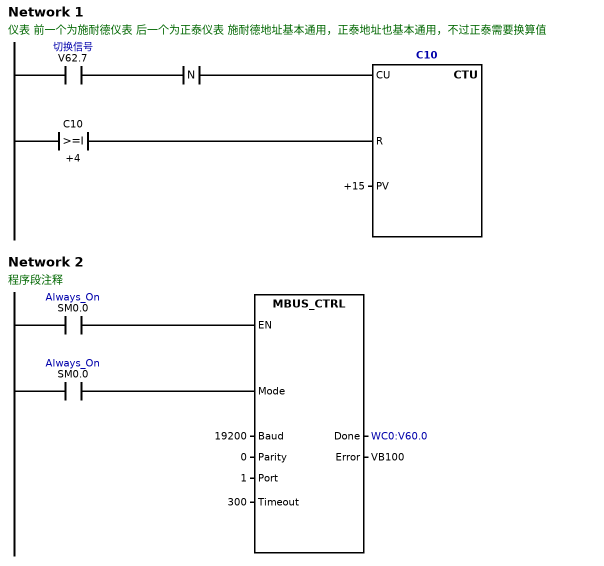
[picture p144: SBR58 networks 1-2]
Network 1
// 仪表 前一个为施耐德仪表 后一个为正泰仪表 施耐德地址基本通用，正泰地址也基本通用，不过正泰需要换算值
LD     切换信号:V62.7
ED
LDW>=  C10, +4
CTU    C10, +15
Network 2
// 程序段注释
LD     Always_On:SM0.0
=      L60.0
LD     Always_On:SM0.0
=      L63.7
LD     L60.0
CALL   MBUS_CTRL:SBR2, L63.7, 19200, 0, 1, 300, WC0:V60.0, VB100
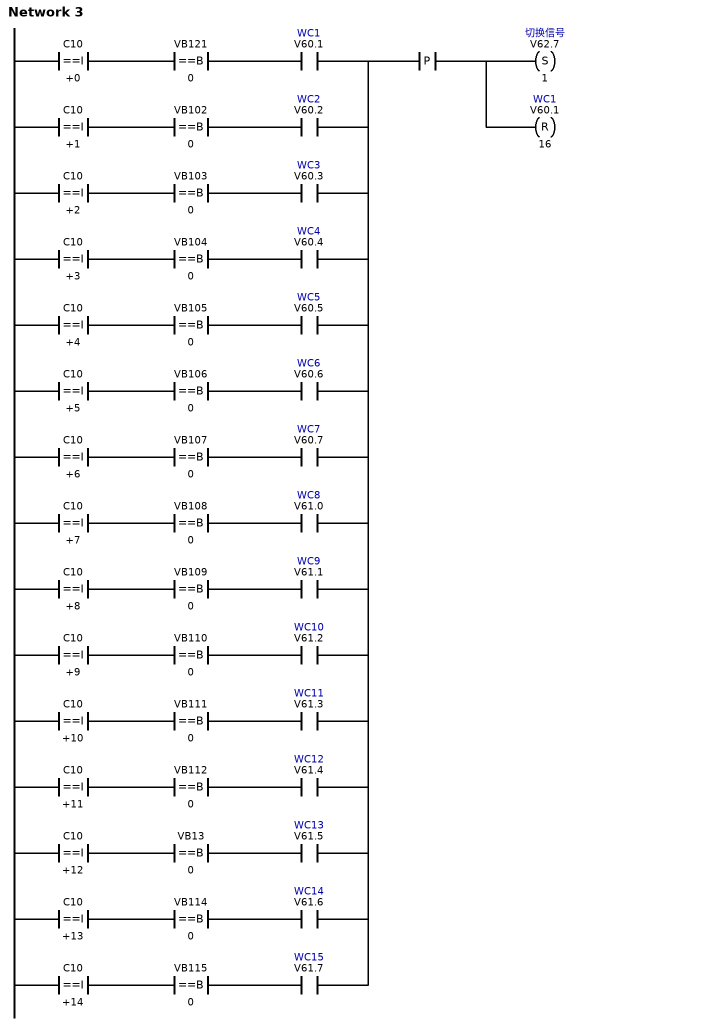
Network 3
LDW=   C10, +0
AB=    VB121, 0
A      WC1:V60.1
LDW=   C10, +1
AB=    VB102, 0
A      WC2:V60.2
OLD
LDW=   C10, +2
AB=    VB103, 0
A      WC3:V60.3
OLD
LDW=   C10, +3
AB=    VB104, 0
A      WC4:V60.4
OLD
LDW=   C10, +4
AB=    VB105, 0
A      WC5:V60.5
OLD
LDW=   C10, +5
AB=    VB106, 0
A      WC6:V60.6
OLD
LDW=   C10, +6
AB=    VB107, 0
A      WC7:V60.7
OLD
LDW=   C10, +7
AB=    VB108, 0
A      WC8:V61.0
OLD
LDW=   C10, +8
AB=    VB109, 0
A      WC9:V61.1
OLD
LDW=   C10, +9
AB=    VB110, 0
A      WC10:V61.2
OLD
LDW=   C10, +10
AB=    VB111, 0
A      WC11:V61.3
OLD
LDW=   C10, +11
AB=    VB112, 0
A      WC12:V61.4
OLD
LDW=   C10, +12
AB=    VB13, 0
A      WC13:V61.5
OLD
LDW=   C10, +13
AB=    VB114, 0
A      WC14:V61.6
OLD
LDW=   C10, +14
AB=    VB115, 0
A      WC15:V61.7
OLD
EU
S      切换信号:V62.7, 1
R      WC1:V60.1, 16
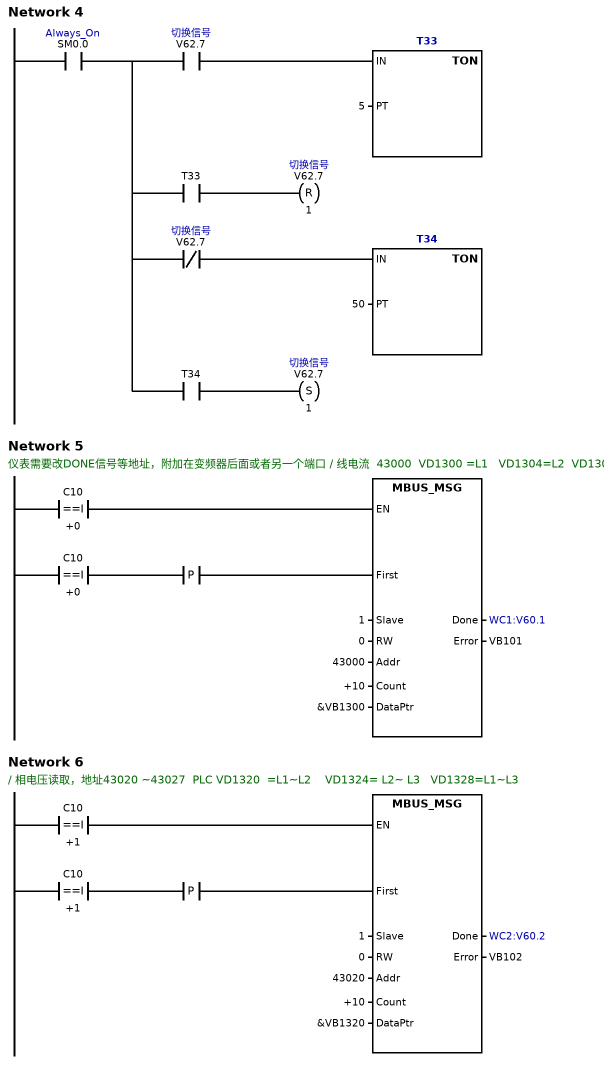
Network 4
LD     Always_On:SM0.0
LPS
A      切换信号:V62.7
TON    T33, 5
LRD
A      T33
R      切换信号:V62.7, 1
LRD
AN     切换信号:V62.7
TON    T34, 50
LPP
A      T34
S      切换信号:V62.7, 1
Network 5
// 仪表需要改DONE信号等地址，附加在变频器后面或者另一个端口
// 线电流  43000  VD1300 =L1   VD1304=L2  VD1308=L3
// 
LDW=   C10, +0
=      L60.0
LDW=   C10, +0
EU
=      L63.7
LD     L60.0
CALL   MBUS_MSG:SBR3, L63.7, 1, 0, 43000, +10, &VB1300, WC1:V60.1, VB101
Network 6
// 
// 相电压读取，地址43020 ~43027  PLC VD1320  =L1~L2    VD1324= L2~ L3   VD1328=L1~L3
LDW=   C10, +1
=      L60.0
LDW=   C10, +1
EU
=      L63.7
LD     L60.0
CALL   MBUS_MSG:SBR3, L63.7, 1, 0, 43020, +10, &VB1320, WC2:V60.2, VB102
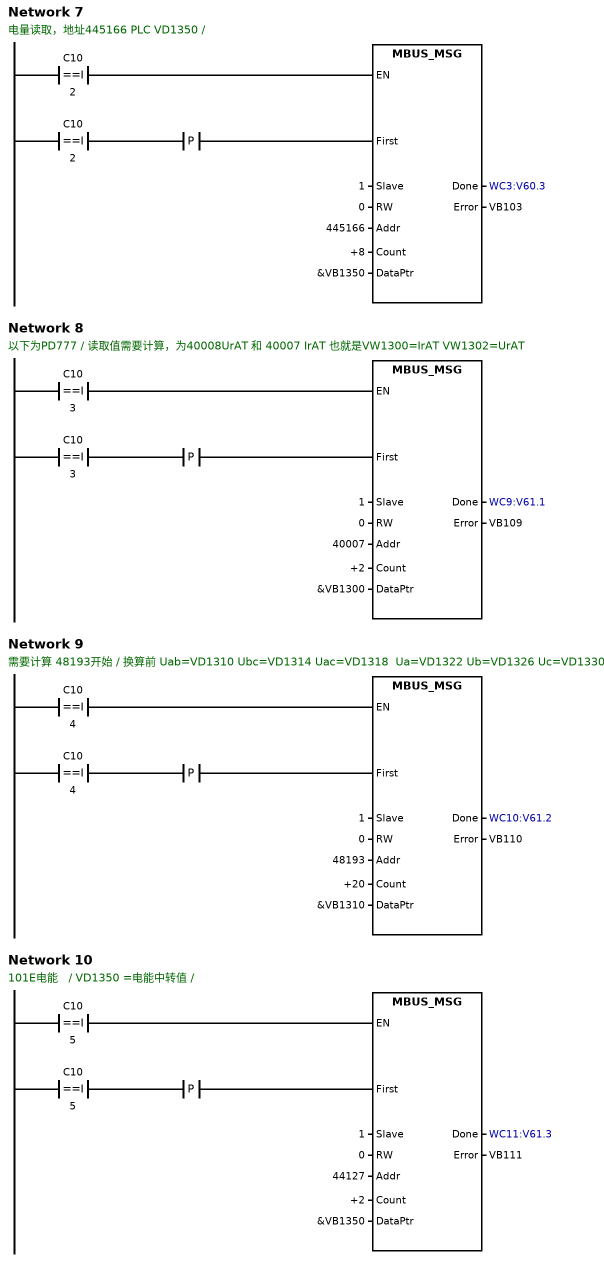
Network 7
// 电量读取，地址445166 PLC VD1350
// 
LDW=   C10, 2
=      L60.0
LDW=   C10, 2
EU
=      L63.7
LD     L60.0
CALL   MBUS_MSG:SBR3, L63.7, 1, 0, 445166, +8, &VB1350, WC3:V60.3, VB103
Network 8
// 以下为PD777
// 读取值需要计算，为40008UrAT 和 40007 IrAT 也就是VW1300=IrAT VW1302=UrAT
LDW=   C10, 3
=      L60.0
LDW=   C10, 3
EU
=      L63.7
LD     L60.0
CALL   MBUS_MSG:SBR3, L63.7, 1, 0, 40007, +2, &VB1300, WC9:V61.1, VB109
Network 9
// 需要计算 48193开始
// 换算前 Uab=VD1310 Ubc=VD1314 Uac=VD1318  Ua=VD1322 Ub=VD1326 Uc=VD1330 
// Ia=VD1334 Ib=VD1338 Ic=VD1342  
// Pt=VD1346 
LDW=   C10, 4
=      L60.0
LDW=   C10, 4
EU
=      L63.7
LD     L60.0
CALL   MBUS_MSG:SBR3, L63.7, 1, 0, 48193, +20, &VB1310, WC10:V61.2, VB110
Network 10
// 101E电能  
// VD1350 =电能中转值
// 
LDW=   C10, 5
=      L60.0
LDW=   C10, 5
EU
=      L63.7
LD     L60.0
CALL   MBUS_MSG:SBR3, L63.7, 1, 0, 44127, +2, &VB1350, WC11:V61.3, VB111
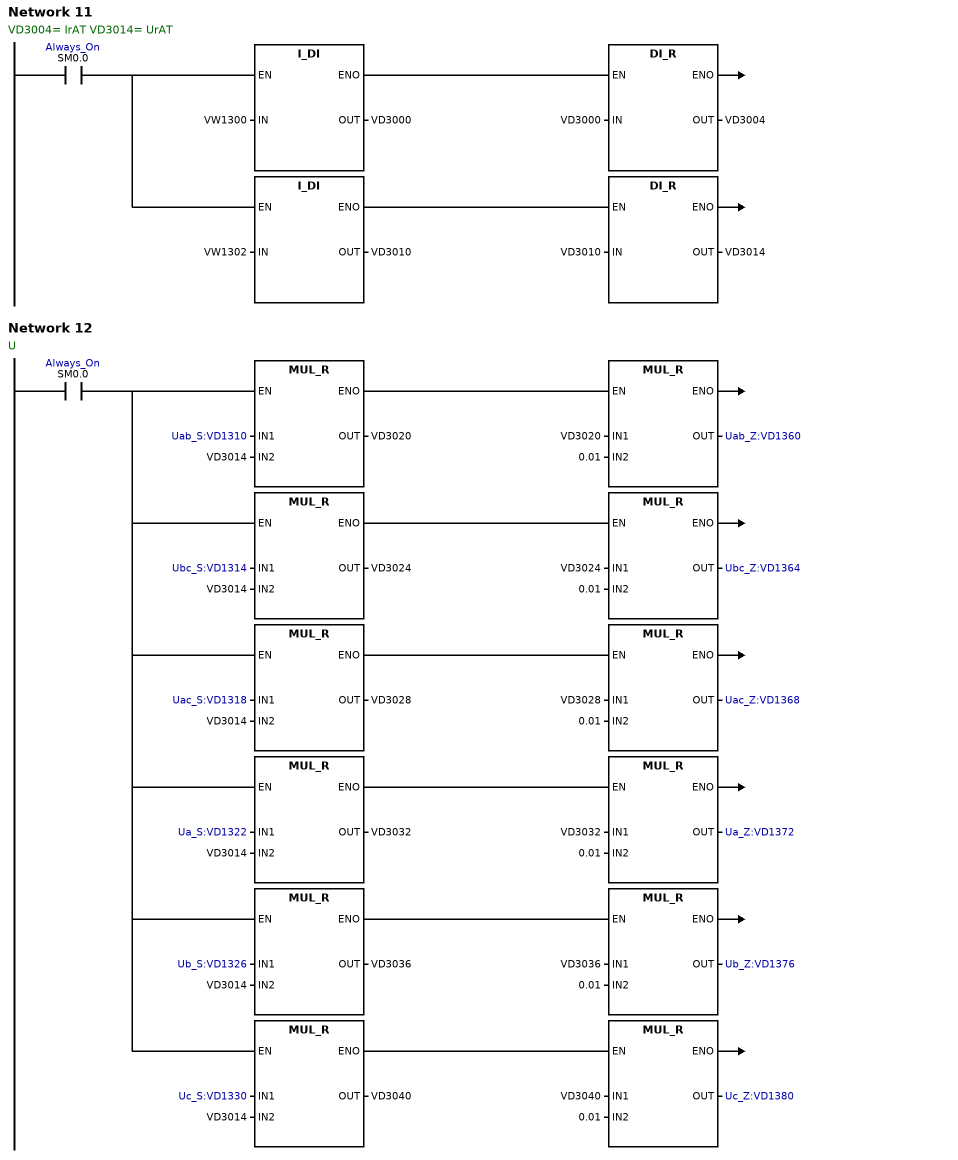
Network 11
// VD3004= IrAT VD3014= UrAT
LD     Always_On:SM0.0
LPS
ITD    VW1300, VD3000
AENO
DTR    VD3000, VD3004
LPP
ITD    VW1302, VD3010
AENO
DTR    VD3010, VD3014
Network 12
// U
LD     Always_On:SM0.0
LPS
MOVR   Uab_S:VD1310, VD3020
AENO
*R     VD3014, VD3020
AENO
MOVR   VD3020, Uab_Z:VD1360
*R     0.01, Uab_Z:VD1360
LRD
MOVR   Ubc_S:VD1314, VD3024
AENO
*R     VD3014, VD3024
AENO
MOVR   VD3024, Ubc_Z:VD1364
*R     0.01, Ubc_Z:VD1364
LRD
MOVR   Uac_S:VD1318, VD3028
AENO
*R     VD3014, VD3028
AENO
MOVR   VD3028, Uac_Z:VD1368
*R     0.01, Uac_Z:VD1368
LRD
MOVR   Ua_S:VD1322, VD3032
AENO
*R     VD3014, VD3032
AENO
MOVR   VD3032, Ua_Z:VD1372
*R     0.01, Ua_Z:VD1372
LRD
MOVR   Ub_S:VD1326, VD3036
AENO
*R     VD3014, VD3036
AENO
MOVR   VD3036, Ub_Z:VD1376
*R     0.01, Ub_Z:VD1376
LPP
MOVR   Uc_S:VD1330, VD3040
AENO
*R     VD3014, VD3040
AENO
MOVR   VD3040, Uc_Z:VD1380
*R     0.01, Uc_Z:VD1380
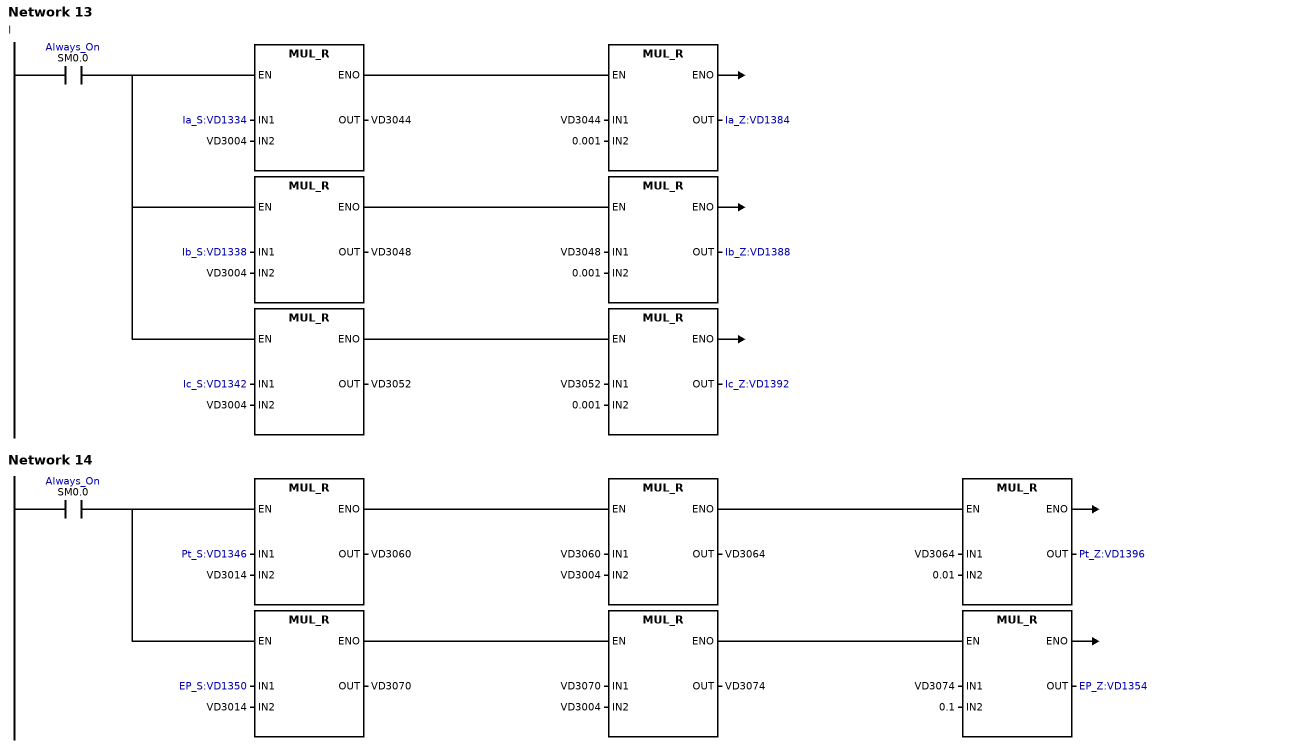
Network 13
// I
LD     Always_On:SM0.0
LPS
MOVR   Ia_S:VD1334, VD3044
AENO
*R     VD3004, VD3044
AENO
MOVR   VD3044, Ia_Z:VD1384
*R     0.001, Ia_Z:VD1384
LRD
MOVR   Ib_S:VD1338, VD3048
AENO
*R     VD3004, VD3048
AENO
MOVR   VD3048, Ib_Z:VD1388
*R     0.001, Ib_Z:VD1388
LPP
MOVR   Ic_S:VD1342, VD3052
AENO
*R     VD3004, VD3052
AENO
MOVR   VD3052, Ic_Z:VD1392
*R     0.001, Ic_Z:VD1392
Network 14
LD     Always_On:SM0.0
LPS
MOVR   Pt_S:VD1346, VD3060
AENO
*R     VD3014, VD3060
AENO
MOVR   VD3060, VD3064
AENO
*R     VD3004, VD3064
AENO
MOVR   VD3064, Pt_Z:VD1396
*R     0.01, Pt_Z:VD1396
LPP
MOVR   EP_S:VD1350, VD3070
AENO
*R     VD3014, VD3070
AENO
MOVR   VD3070, VD3074
AENO
*R     VD3004, VD3074
AENO
MOVR   VD3074, EP_Z:VD1354
*R     0.1, EP_Z:VD1354
END_SUBROUTINE_BLOCK

SUBROUTINE_BLOCK MOD_TCP:SBR60
TITLE=
BEGIN
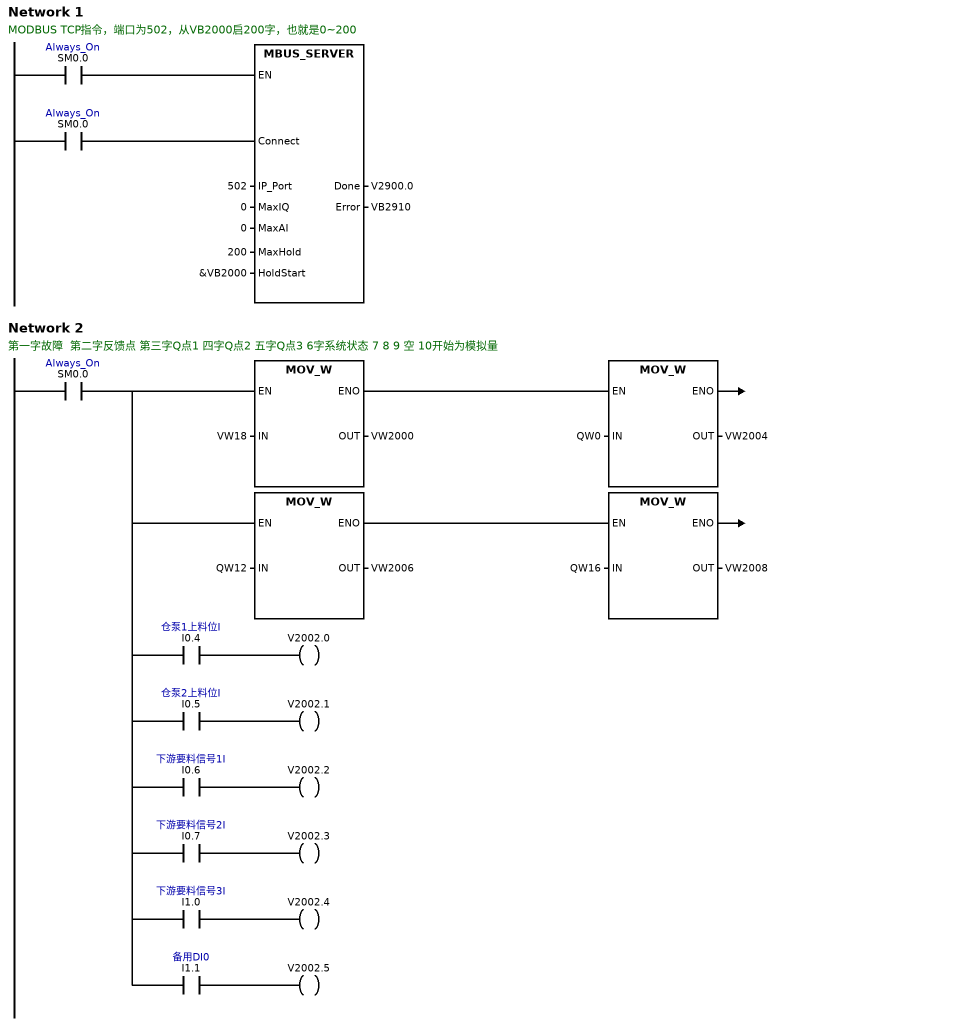
Network 1
// MODBUS TCP指令，端口为502，从VB2000启200字，也就是0~200 
LD     Always_On:SM0.0
=      L60.0
LD     Always_On:SM0.0
=      L63.7
LD     L60.0
CALL   MBUS_SERVER:SBR11, L63.7, 502, 0, 0, 200, &VB2000, V2900.0, VB2910
Network 2
// 第一字故障  第二字反馈点 第三字Q点1 四字Q点2 五字Q点3 6字系统状态 7 8 9 空 10开始为模拟量
LD     Always_On:SM0.0
LPS
MOVW   VW18, VW2000
AENO
MOVW   QW0, VW2004
LRD
MOVW   QW12, VW2006
AENO
MOVW   QW16, VW2008
LRD
A      仓泵1上料位I:I0.4
=      V2002.0
LRD
A      仓泵2上料位I:I0.5
=      V2002.1
LRD
A      下游要料信号1I:I0.6
=      V2002.2
LRD
A      下游要料信号2I:I0.7
=      V2002.3
LRD
A      下游要料信号3I:I1.0
=      V2002.4
LPP
A      备用DI0:I1.1
=      V2002.5
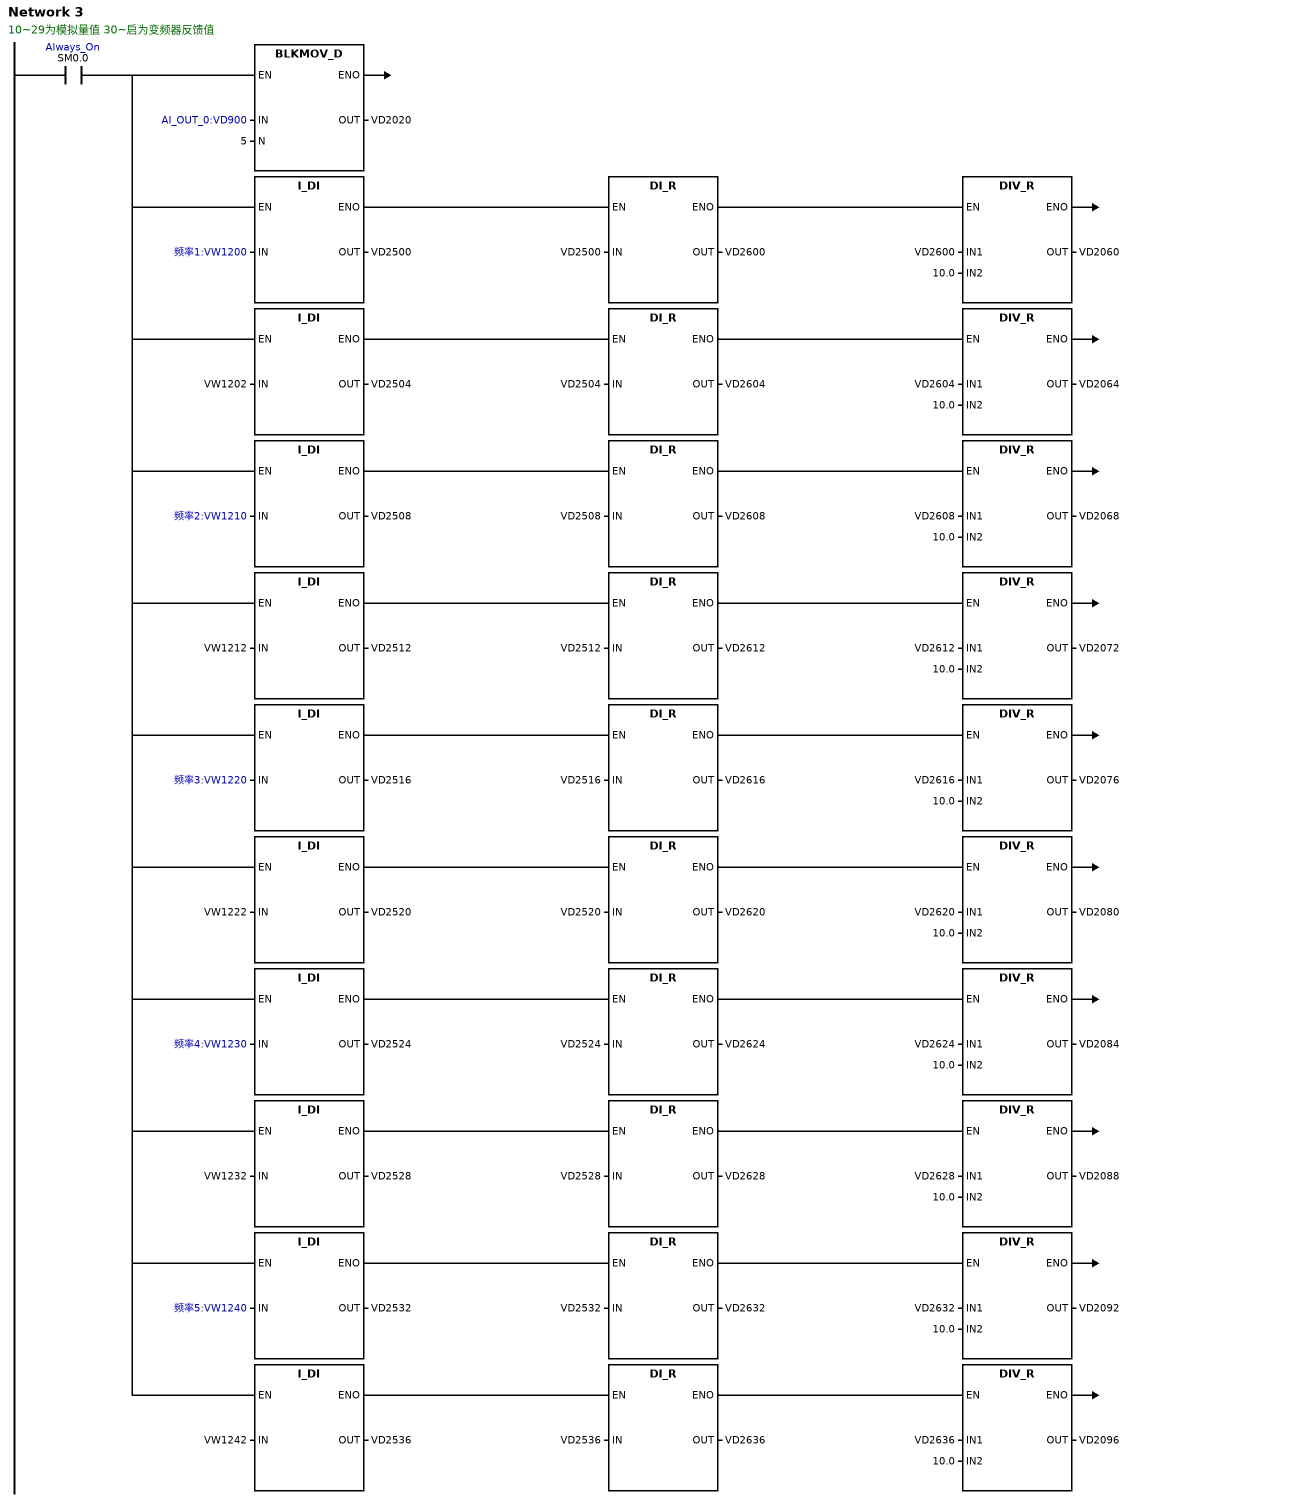
Network 3
// 10~29为模拟量值 30~启为变频器反馈值
LD     Always_On:SM0.0
LPS
BMD    AI_OUT_0:VD900, VD2020, 5
ITD    频率1:VW1200, VD2500
AENO
DTR    VD2500, VD2600
AENO
MOVR   VD2600, VD2060
/R     10.0, VD2060
LRD
ITD    VW1202, VD2504
AENO
DTR    VD2504, VD2604
AENO
MOVR   VD2604, VD2064
/R     10.0, VD2064
LRD
ITD    频率2:VW1210, VD2508
AENO
DTR    VD2508, VD2608
AENO
MOVR   VD2608, VD2068
/R     10.0, VD2068
LRD
ITD    VW1212, VD2512
AENO
DTR    VD2512, VD2612
AENO
MOVR   VD2612, VD2072
/R     10.0, VD2072
LRD
ITD    频率3:VW1220, VD2516
AENO
DTR    VD2516, VD2616
AENO
MOVR   VD2616, VD2076
/R     10.0, VD2076
LRD
ITD    VW1222, VD2520
AENO
DTR    VD2520, VD2620
AENO
MOVR   VD2620, VD2080
/R     10.0, VD2080
LRD
ITD    频率4:VW1230, VD2524
AENO
DTR    VD2524, VD2624
AENO
MOVR   VD2624, VD2084
/R     10.0, VD2084
LRD
ITD    VW1232, VD2528
AENO
DTR    VD2528, VD2628
AENO
MOVR   VD2628, VD2088
/R     10.0, VD2088
LRD
ITD    频率5:VW1240, VD2532
AENO
DTR    VD2532, VD2632
AENO
MOVR   VD2632, VD2092
/R     10.0, VD2092
LPP
ITD    VW1242, VD2536
AENO
DTR    VD2536, VD2636
AENO
MOVR   VD2636, VD2096
/R     10.0, VD2096
END_SUBROUTINE_BLOCK

SUBROUTINE_BLOCK MOD_RTU:SBR61
TITLE=
BEGIN
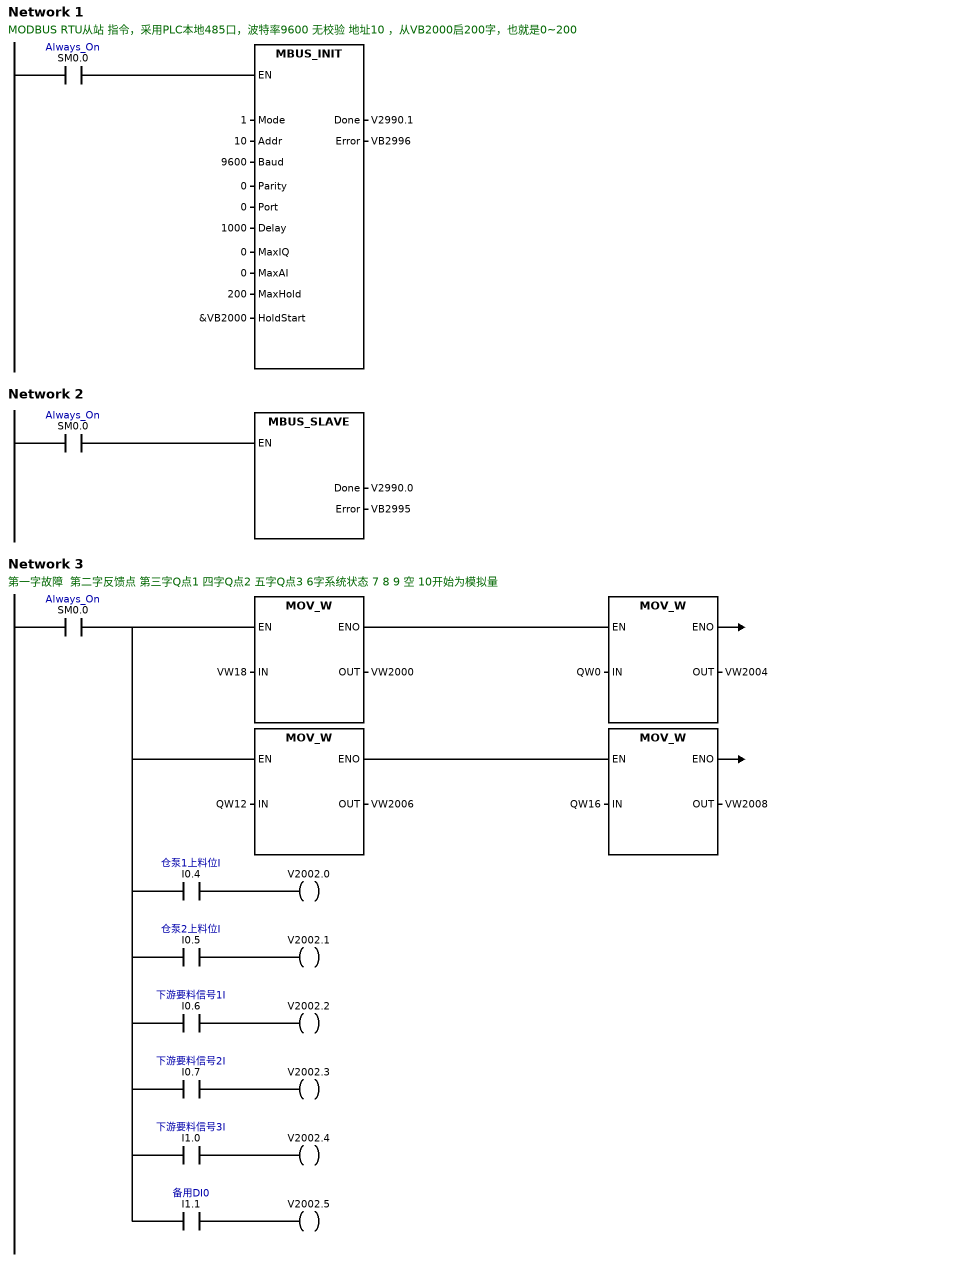
Network 1
// MODBUS RTU从站 指令，采用PLC本地485口，波特率9600 无校验 地址10 ，从VB2000启200字，也就是0~200 
LD     Always_On:SM0.0
CALL   MBUS_INIT:SBR0, 1, 10, 9600, 0, 0, 1000, 0, 0, 200, &VB2000, V2990.1, VB2996
Network 2
LD     Always_On:SM0.0
CALL   MBUS_SLAVE:SBR1, V2990.0, VB2995
Network 3
// 第一字故障  第二字反馈点 第三字Q点1 四字Q点2 五字Q点3 6字系统状态 7 8 9 空 10开始为模拟量
LD     Always_On:SM0.0
LPS
MOVW   VW18, VW2000
AENO
MOVW   QW0, VW2004
LRD
MOVW   QW12, VW2006
AENO
MOVW   QW16, VW2008
LRD
A      仓泵1上料位I:I0.4
=      V2002.0
LRD
A      仓泵2上料位I:I0.5
=      V2002.1
LRD
A      下游要料信号1I:I0.6
=      V2002.2
LRD
A      下游要料信号2I:I0.7
=      V2002.3
LRD
A      下游要料信号3I:I1.0
=      V2002.4
LPP
A      备用DI0:I1.1
=      V2002.5
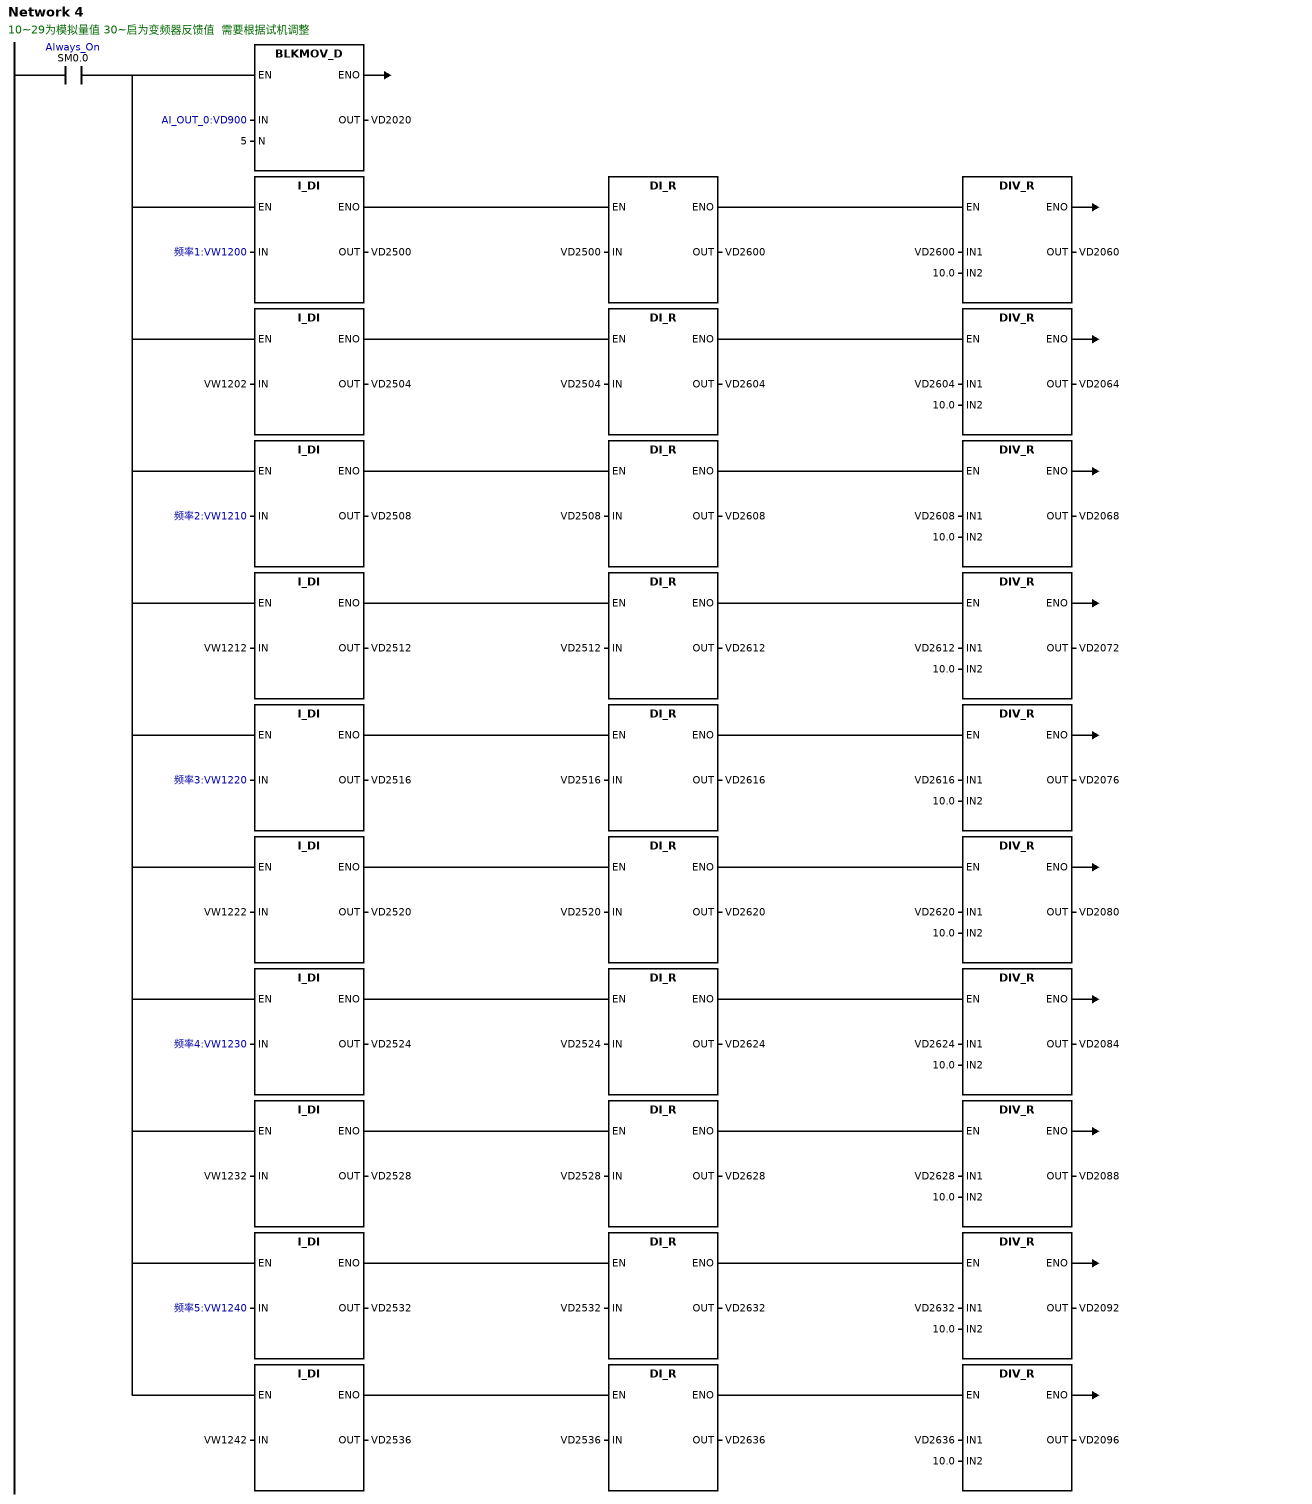
Network 4
// 10~29为模拟量值 30~启为变频器反馈值  需要根据试机调整
LD     Always_On:SM0.0
LPS
BMD    AI_OUT_0:VD900, VD2020, 5
ITD    频率1:VW1200, VD2500
AENO
DTR    VD2500, VD2600
AENO
MOVR   VD2600, VD2060
/R     10.0, VD2060
LRD
ITD    VW1202, VD2504
AENO
DTR    VD2504, VD2604
AENO
MOVR   VD2604, VD2064
/R     10.0, VD2064
LRD
ITD    频率2:VW1210, VD2508
AENO
DTR    VD2508, VD2608
AENO
MOVR   VD2608, VD2068
/R     10.0, VD2068
LRD
ITD    VW1212, VD2512
AENO
DTR    VD2512, VD2612
AENO
MOVR   VD2612, VD2072
/R     10.0, VD2072
LRD
ITD    频率3:VW1220, VD2516
AENO
DTR    VD2516, VD2616
AENO
MOVR   VD2616, VD2076
/R     10.0, VD2076
LRD
ITD    VW1222, VD2520
AENO
DTR    VD2520, VD2620
AENO
MOVR   VD2620, VD2080
/R     10.0, VD2080
LRD
ITD    频率4:VW1230, VD2524
AENO
DTR    VD2524, VD2624
AENO
MOVR   VD2624, VD2084
/R     10.0, VD2084
LRD
ITD    VW1232, VD2528
AENO
DTR    VD2528, VD2628
AENO
MOVR   VD2628, VD2088
/R     10.0, VD2088
LRD
ITD    频率5:VW1240, VD2532
AENO
DTR    VD2532, VD2632
AENO
MOVR   VD2632, VD2092
/R     10.0, VD2092
LPP
ITD    VW1242, VD2536
AENO
DTR    VD2536, VD2636
AENO
MOVR   VD2636, VD2096
/R     10.0, VD2096
END_SUBROUTINE_BLOCK

SUBROUTINE_BLOCK 引风机1:SBR70
TITLE=
VAR_INPUT
IN_SD:BOOL;	// L0.0 
IN_ZD:BOOL;	// L0.1 
IN_Error:BOOL;	// L0.2 
IN_Run_Time:INT;	// LW1 
END_VAR
VAR_OUTPUT
OUT_主:BOOL;	// L3.0  先主
OUT_角:BOOL;	// L3.1 后角
OUT_星:BOOL;	// L3.2 先星
END_VAR
VAR
TP1:BOOL;	// L3.3 
TP2:BOOL;	// L3.4 
END_VAR
BEGIN
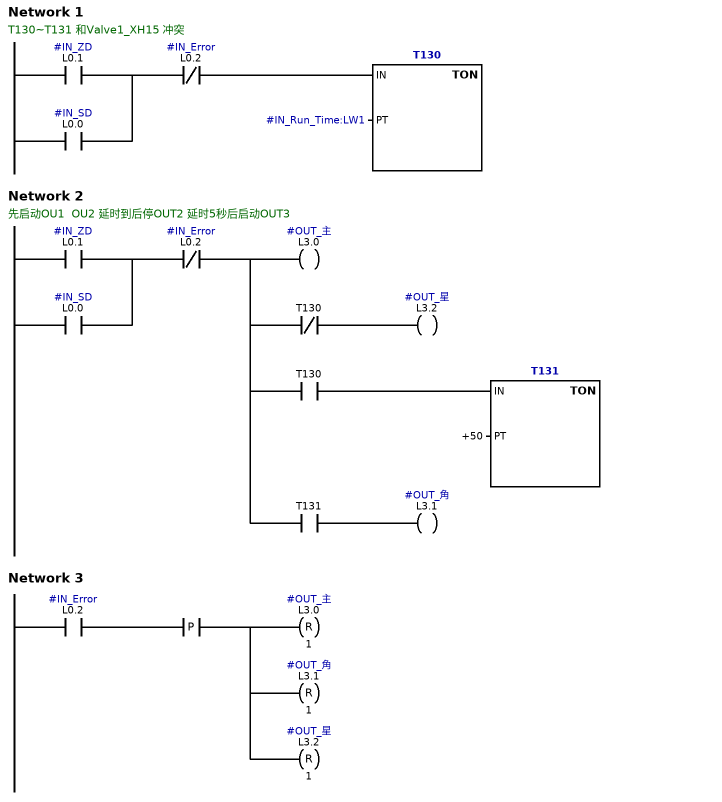
Network 1
// T130~T131 和Valve1_XH15 冲突
LD     #IN_ZD:L0.1
O      #IN_SD:L0.0
AN     #IN_Error:L0.2
TON    T130, #IN_Run_Time:LW1
Network 2
// 先启动OU1  OU2 延时到后停OUT2 延时5秒后启动OUT3
LD     #IN_ZD:L0.1
O      #IN_SD:L0.0
AN     #IN_Error:L0.2
LPS
=      #OUT_主:L3.0
AN     T130
=      #OUT_星:L3.2
LRD
A      T130
TON    T131, +50
LPP
A      T131
=      #OUT_角:L3.1
Network 3
LD     #IN_Error:L0.2
EU
R      #OUT_主:L3.0, 1
R      #OUT_角:L3.1, 1
R      #OUT_星:L3.2, 1
END_SUBROUTINE_BLOCK

SUBROUTINE_BLOCK 引风机2:SBR71
TITLE=
VAR_INPUT
IN_SD:BOOL;	// L0.0 
IN_ZD:BOOL;	// L0.1 
IN_Error:BOOL;	// L0.2 
IN_Run_Time:INT;	// LW1 
END_VAR
VAR_OUTPUT
OUT_ONE1:BOOL;	// L3.0 
OUT_ONE2:BOOL;	// L3.1 
OUT_ONE3:BOOL;	// L3.2 
END_VAR
VAR
TP1:BOOL;	// L3.3 
TP2:BOOL;	// L3.4 
END_VAR
BEGIN
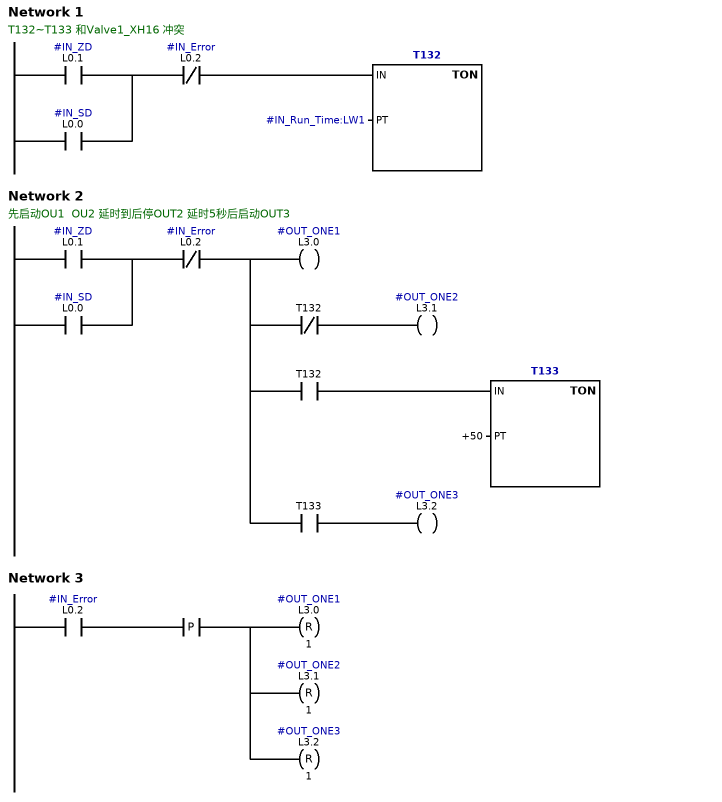
Network 1
// T132~T133 和Valve1_XH16 冲突
LD     #IN_ZD:L0.1
O      #IN_SD:L0.0
AN     #IN_Error:L0.2
TON    T132, #IN_Run_Time:LW1
Network 2
// 先启动OU1  OU2 延时到后停OUT2 延时5秒后启动OUT3
LD     #IN_ZD:L0.1
O      #IN_SD:L0.0
AN     #IN_Error:L0.2
LPS
=      #OUT_ONE1:L3.0
AN     T132
=      #OUT_ONE2:L3.1
LRD
A      T132
TON    T133, +50
LPP
A      T133
=      #OUT_ONE3:L3.2
Network 3
LD     #IN_Error:L0.2
EU
R      #OUT_ONE1:L3.0, 1
R      #OUT_ONE2:L3.1, 1
R      #OUT_ONE3:L3.2, 1
END_SUBROUTINE_BLOCK

SUBROUTINE_BLOCK 引风机3:SBR72
TITLE=
VAR_INPUT
IN_SD:BOOL;	// L0.0 
IN_ZD:BOOL;	// L0.1 
IN_Error:BOOL;	// L0.2 
IN_Run_Time:INT;	// LW1 
END_VAR
VAR_OUTPUT
OUT_ONE1:BOOL;	// L3.0 
OUT_ONE2:BOOL;	// L3.1 
OUT_ONE3:BOOL;	// L3.2 
END_VAR
VAR
TP1:BOOL;	// L3.3 
TP2:BOOL;	// L3.4 
END_VAR
BEGIN
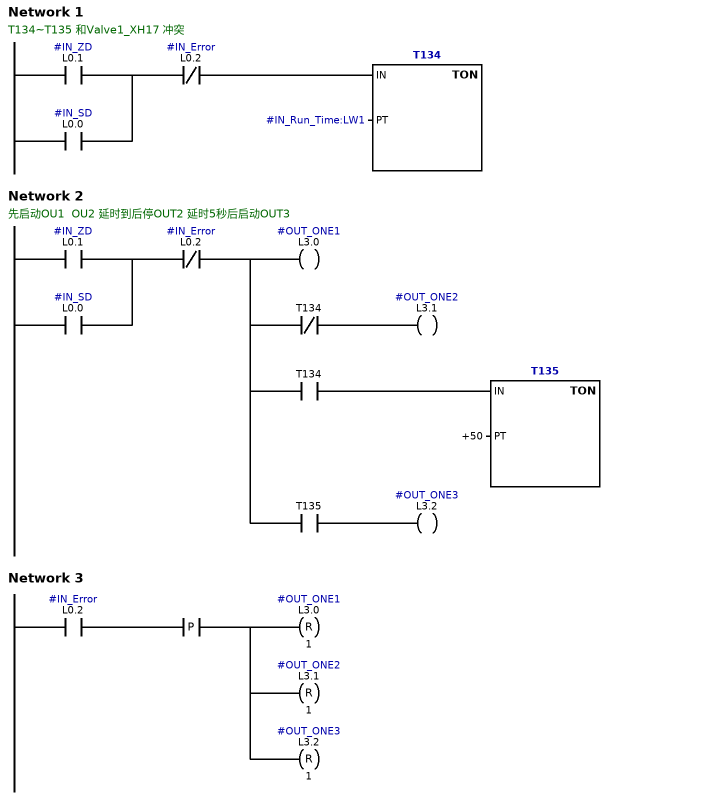
Network 1
// T134~T135 和Valve1_XH17 冲突
LD     #IN_ZD:L0.1
O      #IN_SD:L0.0
AN     #IN_Error:L0.2
TON    T134, #IN_Run_Time:LW1
Network 2
// 先启动OU1  OU2 延时到后停OUT2 延时5秒后启动OUT3
LD     #IN_ZD:L0.1
O      #IN_SD:L0.0
AN     #IN_Error:L0.2
LPS
=      #OUT_ONE1:L3.0
AN     T134
=      #OUT_ONE2:L3.1
LRD
A      T134
TON    T135, +50
LPP
A      T135
=      #OUT_ONE3:L3.2
Network 3
LD     #IN_Error:L0.2
EU
R      #OUT_ONE1:L3.0, 1
R      #OUT_ONE2:L3.1, 1
R      #OUT_ONE3:L3.2, 1
END_SUBROUTINE_BLOCK

SUBROUTINE_BLOCK 引风机4:SBR73
TITLE=
VAR_INPUT
IN_SD:BOOL;	// L0.0 
IN_ZD:BOOL;	// L0.1 
IN_Error:BOOL;	// L0.2 
IN_Run_Time:INT;	// LW1 
END_VAR
VAR_OUTPUT
OUT_ONE1:BOOL;	// L3.0 
OUT_ONE2:BOOL;	// L3.1 
OUT_ONE3:BOOL;	// L3.2 
END_VAR
VAR
TP1:BOOL;	// L3.3 
TP2:BOOL;	// L3.4 
END_VAR
BEGIN
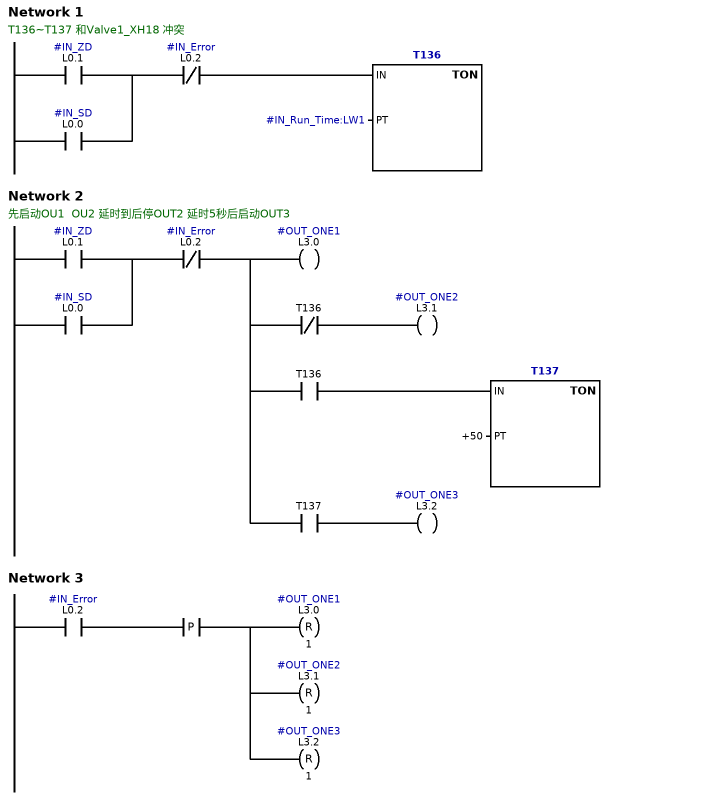
Network 1
// T136~T137 和Valve1_XH18 冲突
LD     #IN_ZD:L0.1
O      #IN_SD:L0.0
AN     #IN_Error:L0.2
TON    T136, #IN_Run_Time:LW1
Network 2
// 先启动OU1  OU2 延时到后停OUT2 延时5秒后启动OUT3
LD     #IN_ZD:L0.1
O      #IN_SD:L0.0
AN     #IN_Error:L0.2
LPS
=      #OUT_ONE1:L3.0
AN     T136
=      #OUT_ONE2:L3.1
LRD
A      T136
TON    T137, +50
LPP
A      T137
=      #OUT_ONE3:L3.2
Network 3
LD     #IN_Error:L0.2
EU
R      #OUT_ONE1:L3.0, 1
R      #OUT_ONE2:L3.1, 1
R      #OUT_ONE3:L3.2, 1
END_SUBROUTINE_BLOCK

SUBROUTINE_BLOCK 引风机5:SBR74
TITLE=
VAR_INPUT
IN_SD:BOOL;	// L0.0 
IN_ZD:BOOL;	// L0.1 
IN_Error:BOOL;	// L0.2 
IN_Run_Time:INT;	// LW1 
END_VAR
VAR_OUTPUT
OUT_ONE1:BOOL;	// L3.0 
OUT_ONE2:BOOL;	// L3.1 
OUT_ONE3:BOOL;	// L3.2 
END_VAR
VAR
TP1:BOOL;	// L3.3 
TP2:BOOL;	// L3.4 
END_VAR
BEGIN
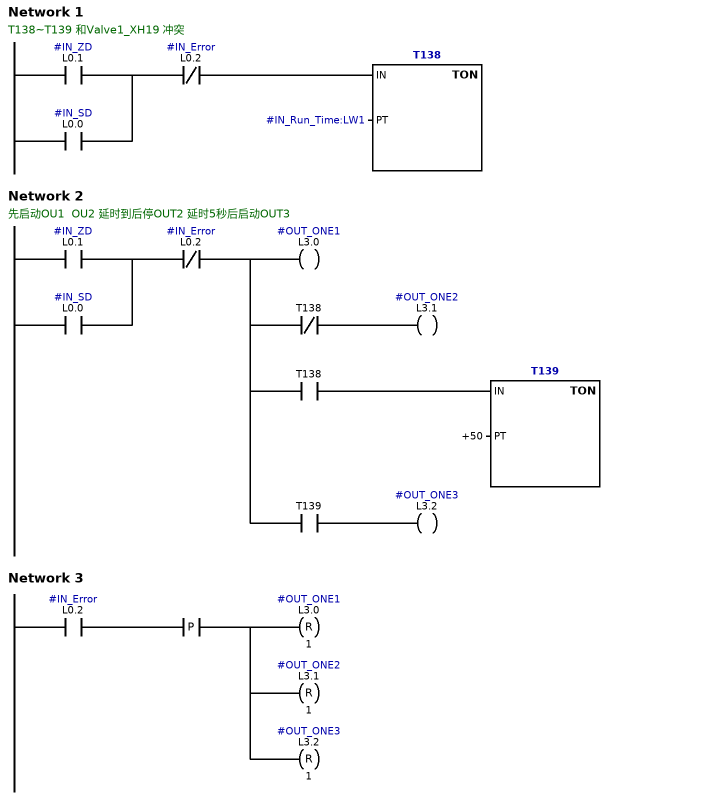
Network 1
// T138~T139 和Valve1_XH19 冲突
LD     #IN_ZD:L0.1
O      #IN_SD:L0.0
AN     #IN_Error:L0.2
TON    T138, #IN_Run_Time:LW1
Network 2
// 先启动OU1  OU2 延时到后停OUT2 延时5秒后启动OUT3
LD     #IN_ZD:L0.1
O      #IN_SD:L0.0
AN     #IN_Error:L0.2
LPS
=      #OUT_ONE1:L3.0
AN     T138
=      #OUT_ONE2:L3.1
LRD
A      T138
TON    T139, +50
LPP
A      T139
=      #OUT_ONE3:L3.2
Network 3
LD     #IN_Error:L0.2
EU
R      #OUT_ONE1:L3.0, 1
R      #OUT_ONE2:L3.1, 1
R      #OUT_ONE3:L3.2, 1
END_SUBROUTINE_BLOCK

SUBROUTINE_BLOCK 除铁器6组4:SBR76
TITLE=
VAR_INPUT
IN_SD:BOOL;	// L0.0 
IN_ZD:BOOL;	// L0.1 
IN_Error:BOOL;	// L0.2 
IN_Run_Time:INT;	// LW1 
IN_Stop_Time:INT;	// LW3 
IN_JG:INT;	// LW5 除铁到排渣间隔
IN_PZ_RT:INT;	// LW7 排渣运行
IN_PZ_ST:INT;	// LW9 排渣间隔
Z_Time:DINT;	// LD11 
END_VAR
VAR_OUTPUT
OUT_1:BOOL;	// L15.0 
OUT_2:BOOL;	// L15.1 
OUT_3:BOOL;	// L15.2 
OUT_4:BOOL;	// L15.3 
OUT_5:BOOL;	// L15.4 
OUT_6:BOOL;	// L15.5 
ZTXH:BOOL;	// L15.6 暂停信号
END_VAR
BEGIN
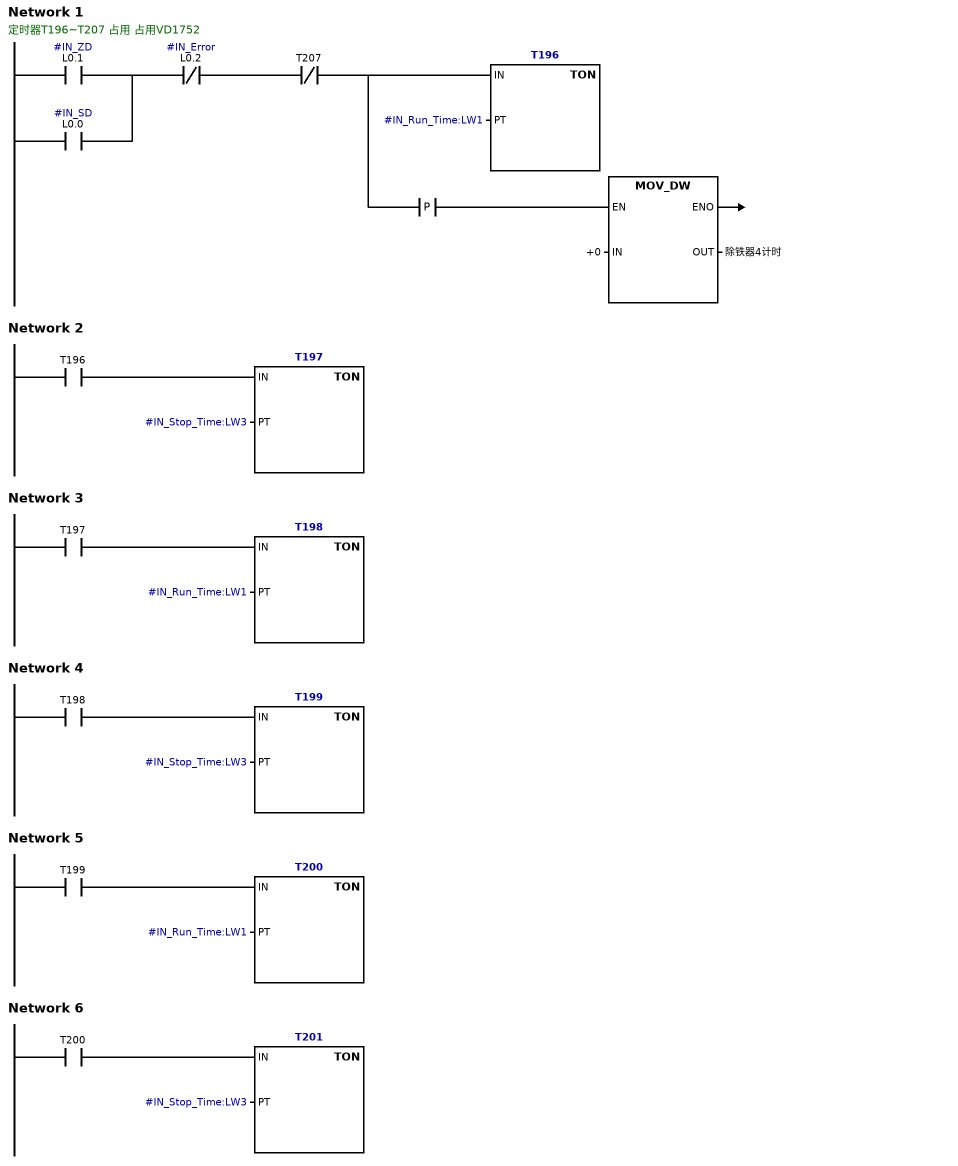
Network 1
// 定时器T196~T207 占用 占用VD1752
// (network saved uncompiled; LAD cells follow)
// row 0: c0 -| |- #IN_ZD:L0.1 v  c1 -|/|- #IN_Error:L0.2  c2 -|/|- T207 v  c3 --  c4 [TON T196 IN:=power@row0, PT:=#IN_Run_Time:LW1]
// row 1: c0 -| |- #IN_SD:L0.0 ^  c2 ^v  c4 [box]
// row 2: c2 ^  c3 -|P|-  c4 --  c5 [MOV_DW EN:=power@row2, IN:=+0, ENO=>power, OUT=>除铁器4计时]  c6 ->
// row 3: c5 [box]
Network 2
LD     T196
TON    T197, #IN_Stop_Time:LW3
Network 3
LD     T197
TON    T198, #IN_Run_Time:LW1
Network 4
LD     T198
TON    T199, #IN_Stop_Time:LW3
Network 5
LD     T199
TON    T200, #IN_Run_Time:LW1
Network 6
LD     T200
TON    T201, #IN_Stop_Time:LW3
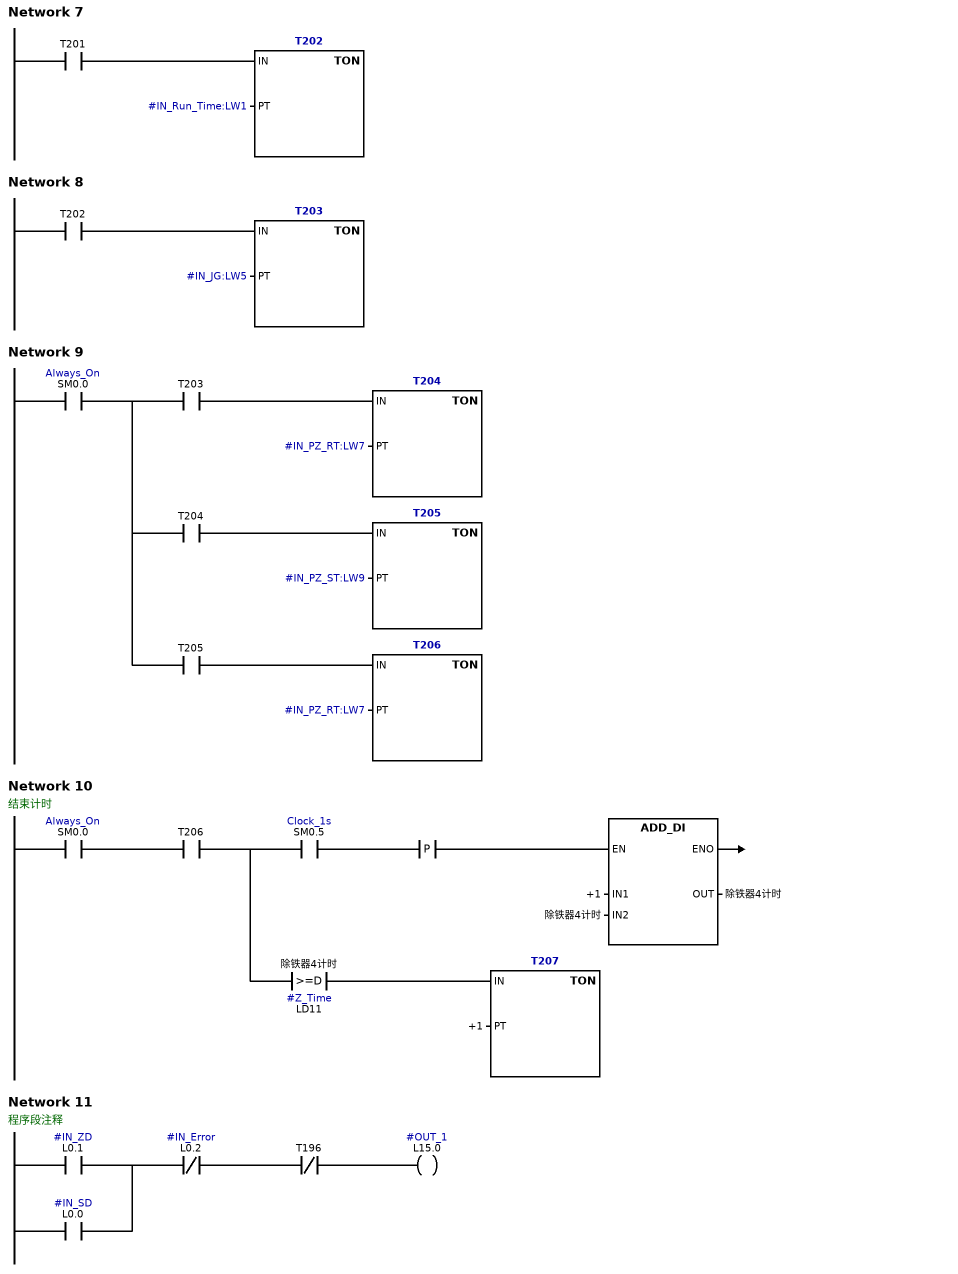
Network 7
LD     T201
TON    T202, #IN_Run_Time:LW1
Network 8
LD     T202
TON    T203, #IN_JG:LW5
Network 9
LD     Always_On:SM0.0
LPS
A      T203
TON    T204, #IN_PZ_RT:LW7
LRD
A      T204
TON    T205, #IN_PZ_ST:LW9
LPP
A      T205
TON    T206, #IN_PZ_RT:LW7
Network 10
// 结束计时
// (network saved uncompiled; LAD cells follow)
// row 0: c0 -| |- Always_On:SM0.0  c1 -| |- T206 v  c2 -| |- Clock_1s:SM0.5  c3 -|P|-  c4 --  c5 [ADD_DI EN:=power@row0, IN1:=+1, IN2:=除铁器4计时, ENO=>power, OUT=>除铁器4计时]  c6 ->
// row 1: c1 ^v  c5 [box]
// row 2: c1 ^  c2 -|>=D|- 除铁器4计时, #Z_Time:LD11  c3 --  c4 [TON T207 IN:=power@row2, PT:=+1]
// row 3: c4 [box]
Network 11
//  程序段注释
LD     #IN_ZD:L0.1
O      #IN_SD:L0.0
AN     #IN_Error:L0.2
AN     T196
=      #OUT_1:L15.0
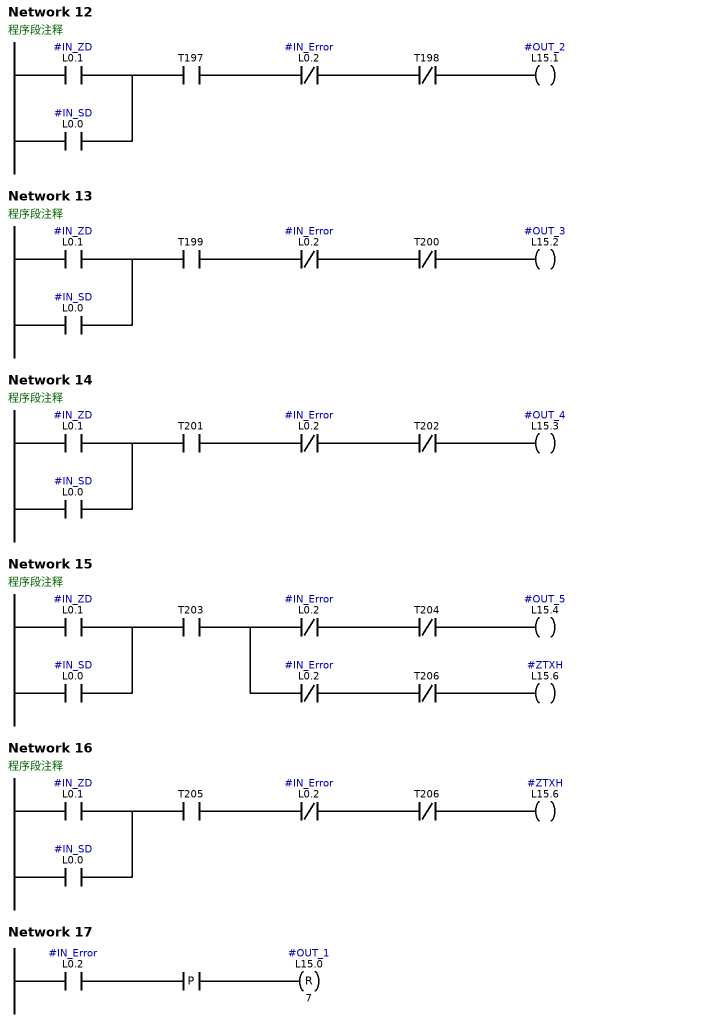
Network 12
//  程序段注释
LD     #IN_ZD:L0.1
O      #IN_SD:L0.0
A      T197
AN     #IN_Error:L0.2
AN     T198
=      #OUT_2:L15.1
Network 13
//  程序段注释
LD     #IN_ZD:L0.1
O      #IN_SD:L0.0
A      T199
AN     #IN_Error:L0.2
AN     T200
=      #OUT_3:L15.2
Network 14
//  程序段注释
LD     #IN_ZD:L0.1
O      #IN_SD:L0.0
A      T201
AN     #IN_Error:L0.2
AN     T202
=      #OUT_4:L15.3
Network 15
//  程序段注释
LD     #IN_ZD:L0.1
O      #IN_SD:L0.0
A      T203
LPS
AN     #IN_Error:L0.2
AN     T204
=      #OUT_5:L15.4
LPP
AN     #IN_Error:L0.2
AN     T206
=      #ZTXH:L15.6
Network 16
//  程序段注释
LD     #IN_ZD:L0.1
O      #IN_SD:L0.0
A      T205
AN     #IN_Error:L0.2
AN     T206
=      #ZTXH:L15.6
Network 17
LD     #IN_Error:L0.2
EU
R      #OUT_1:L15.0, 7
END_SUBROUTINE_BLOCK

SUBROUTINE_BLOCK 除铁器6组1:SBR77
TITLE=
VAR_INPUT
IN_SD:BOOL;	// L0.0 
IN_ZD:BOOL;	// L0.1 
IN_Error:BOOL;	// L0.2 
IN_Run_Time:INT;	// LW1 
IN_Stop_Time:INT;	// LW3 
IN_JG:INT;	// LW5 除铁到排渣间隔
IN_PZ_RT:INT;	// LW7 排渣运行
IN_PZ_ST:INT;	// LW9 排渣间隔
Z_Time:DINT;	// LD11 
END_VAR
VAR_OUTPUT
OUT_1:BOOL;	// L15.0 
OUT_2:BOOL;	// L15.1 
OUT_3:BOOL;	// L15.2 
OUT_4:BOOL;	// L15.3 
OUT_5:BOOL;	// L15.4 
OUT_6:BOOL;	// L15.5 
ZTXH:BOOL;	// L15.6 暂停信号
END_VAR
BEGIN
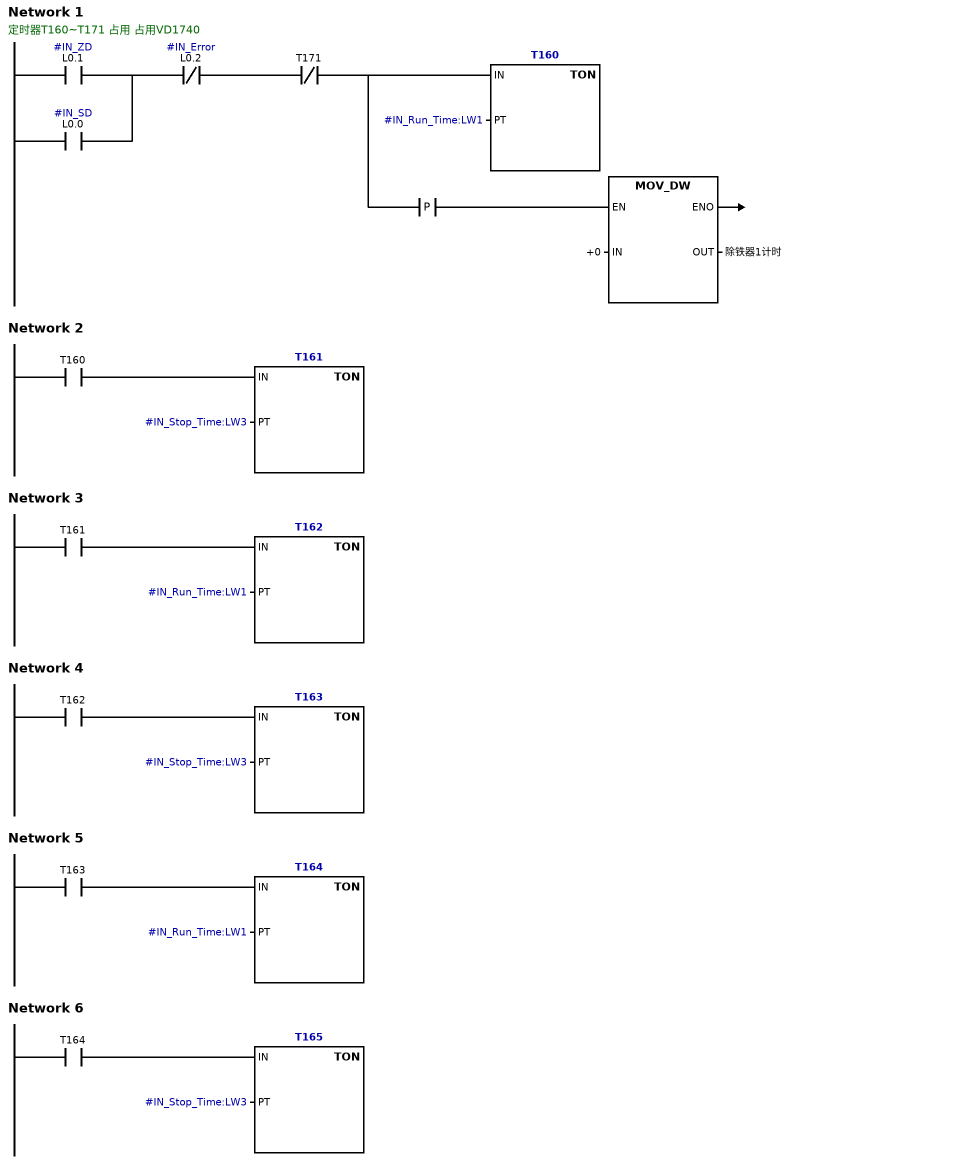
Network 1
// 定时器T160~T171 占用 占用VD1740
// (network saved uncompiled; LAD cells follow)
// row 0: c0 -| |- #IN_ZD:L0.1 v  c1 -|/|- #IN_Error:L0.2  c2 -|/|- T171 v  c3 --  c4 [TON T160 IN:=power@row0, PT:=#IN_Run_Time:LW1]
// row 1: c0 -| |- #IN_SD:L0.0 ^  c2 ^v  c4 [box]
// row 2: c2 ^  c3 -|P|-  c4 --  c5 [MOV_DW EN:=power@row2, IN:=+0, ENO=>power, OUT=>除铁器1计时]  c6 ->
// row 3: c5 [box]
Network 2
LD     T160
TON    T161, #IN_Stop_Time:LW3
Network 3
LD     T161
TON    T162, #IN_Run_Time:LW1
Network 4
LD     T162
TON    T163, #IN_Stop_Time:LW3
Network 5
LD     T163
TON    T164, #IN_Run_Time:LW1
Network 6
LD     T164
TON    T165, #IN_Stop_Time:LW3
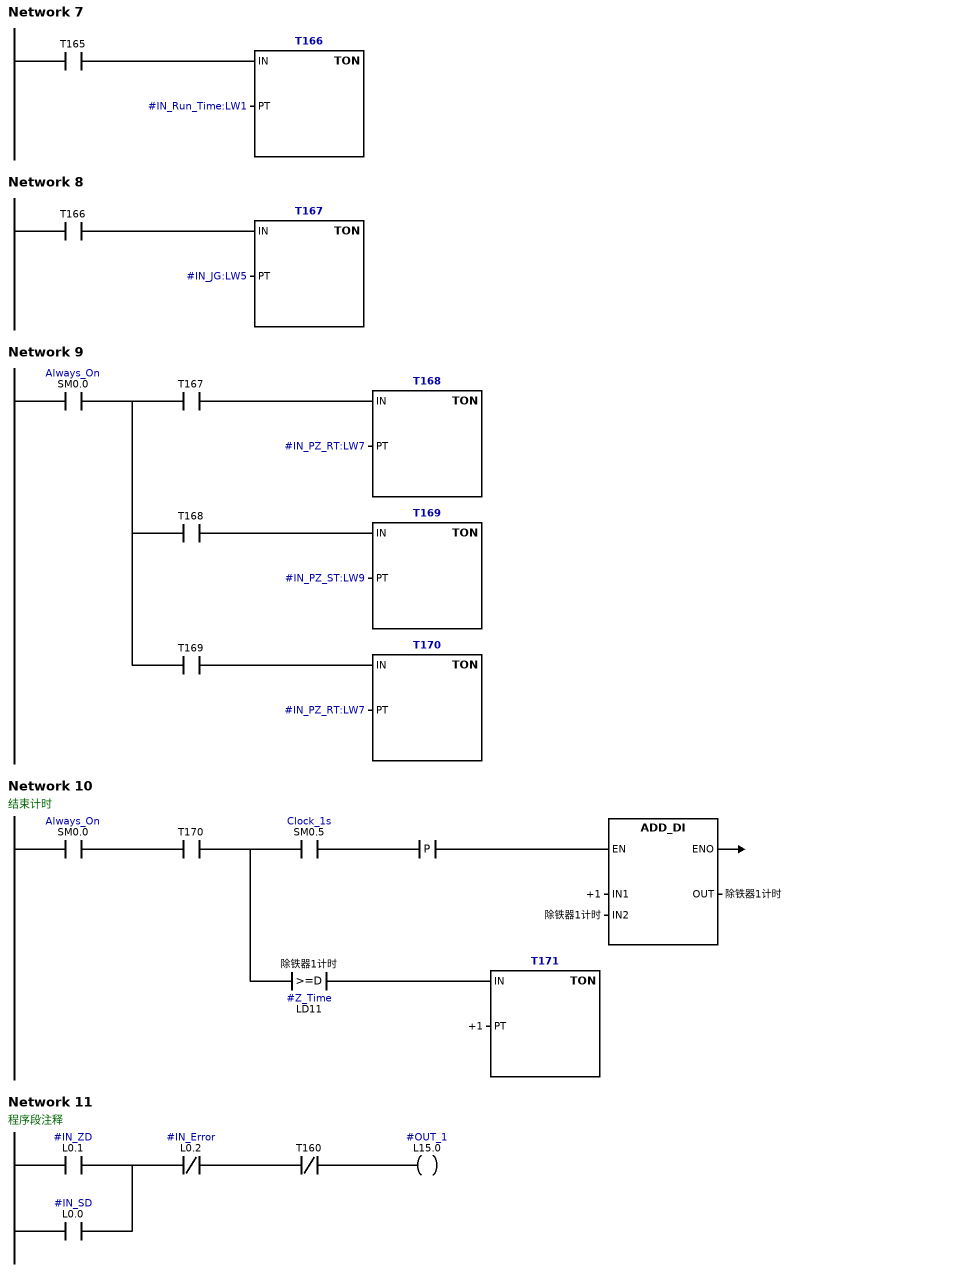
Network 7
LD     T165
TON    T166, #IN_Run_Time:LW1
Network 8
LD     T166
TON    T167, #IN_JG:LW5
Network 9
LD     Always_On:SM0.0
LPS
A      T167
TON    T168, #IN_PZ_RT:LW7
LRD
A      T168
TON    T169, #IN_PZ_ST:LW9
LPP
A      T169
TON    T170, #IN_PZ_RT:LW7
Network 10
// 结束计时
// (network saved uncompiled; LAD cells follow)
// row 0: c0 -| |- Always_On:SM0.0  c1 -| |- T170 v  c2 -| |- Clock_1s:SM0.5  c3 -|P|-  c4 --  c5 [ADD_DI EN:=power@row0, IN1:=+1, IN2:=除铁器1计时, ENO=>power, OUT=>除铁器1计时]  c6 ->
// row 1: c1 ^v  c5 [box]
// row 2: c1 ^  c2 -|>=D|- 除铁器1计时, #Z_Time:LD11  c3 --  c4 [TON T171 IN:=power@row2, PT:=+1]
// row 3: c4 [box]
Network 11
//  程序段注释
LD     #IN_ZD:L0.1
O      #IN_SD:L0.0
AN     #IN_Error:L0.2
AN     T160
=      #OUT_1:L15.0
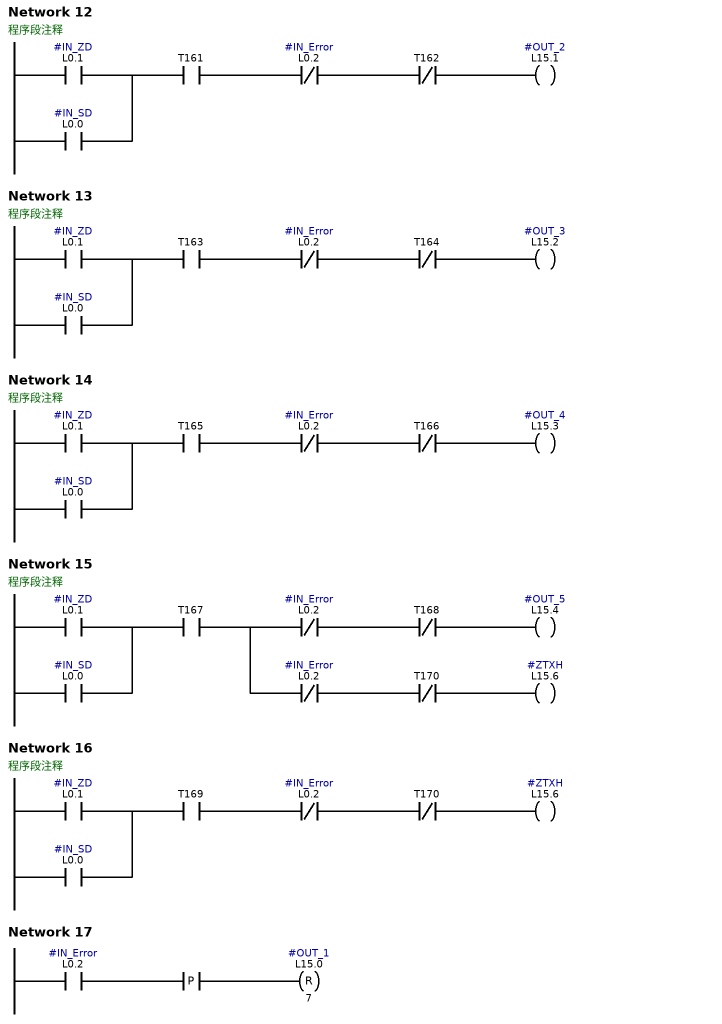
Network 12
//  程序段注释
LD     #IN_ZD:L0.1
O      #IN_SD:L0.0
A      T161
AN     #IN_Error:L0.2
AN     T162
=      #OUT_2:L15.1
Network 13
//  程序段注释
LD     #IN_ZD:L0.1
O      #IN_SD:L0.0
A      T163
AN     #IN_Error:L0.2
AN     T164
=      #OUT_3:L15.2
Network 14
//  程序段注释
LD     #IN_ZD:L0.1
O      #IN_SD:L0.0
A      T165
AN     #IN_Error:L0.2
AN     T166
=      #OUT_4:L15.3
Network 15
//  程序段注释
LD     #IN_ZD:L0.1
O      #IN_SD:L0.0
A      T167
LPS
AN     #IN_Error:L0.2
AN     T168
=      #OUT_5:L15.4
LPP
AN     #IN_Error:L0.2
AN     T170
=      #ZTXH:L15.6
Network 16
//  程序段注释
LD     #IN_ZD:L0.1
O      #IN_SD:L0.0
A      T169
AN     #IN_Error:L0.2
AN     T170
=      #ZTXH:L15.6
Network 17
LD     #IN_Error:L0.2
EU
R      #OUT_1:L15.0, 7
END_SUBROUTINE_BLOCK

SUBROUTINE_BLOCK 除铁器6组2:SBR78
TITLE=
VAR_INPUT
IN_SD:BOOL;	// L0.0 
IN_ZD:BOOL;	// L0.1 
IN_Error:BOOL;	// L0.2 
IN_Run_Time:INT;	// LW1 
IN_Stop_Time:INT;	// LW3 
IN_JG:INT;	// LW5 除铁到排渣间隔
IN_PZ_RT:INT;	// LW7 排渣运行
IN_PZ_ST:INT;	// LW9 排渣间隔
Z_Time:DINT;	// LD11 
END_VAR
VAR_OUTPUT
OUT_1:BOOL;	// L15.0 
OUT_2:BOOL;	// L15.1 
OUT_3:BOOL;	// L15.2 
OUT_4:BOOL;	// L15.3 
OUT_5:BOOL;	// L15.4 
OUT_6:BOOL;	// L15.5 
ZTXH:BOOL;	// L15.6 暂停信号
END_VAR
BEGIN
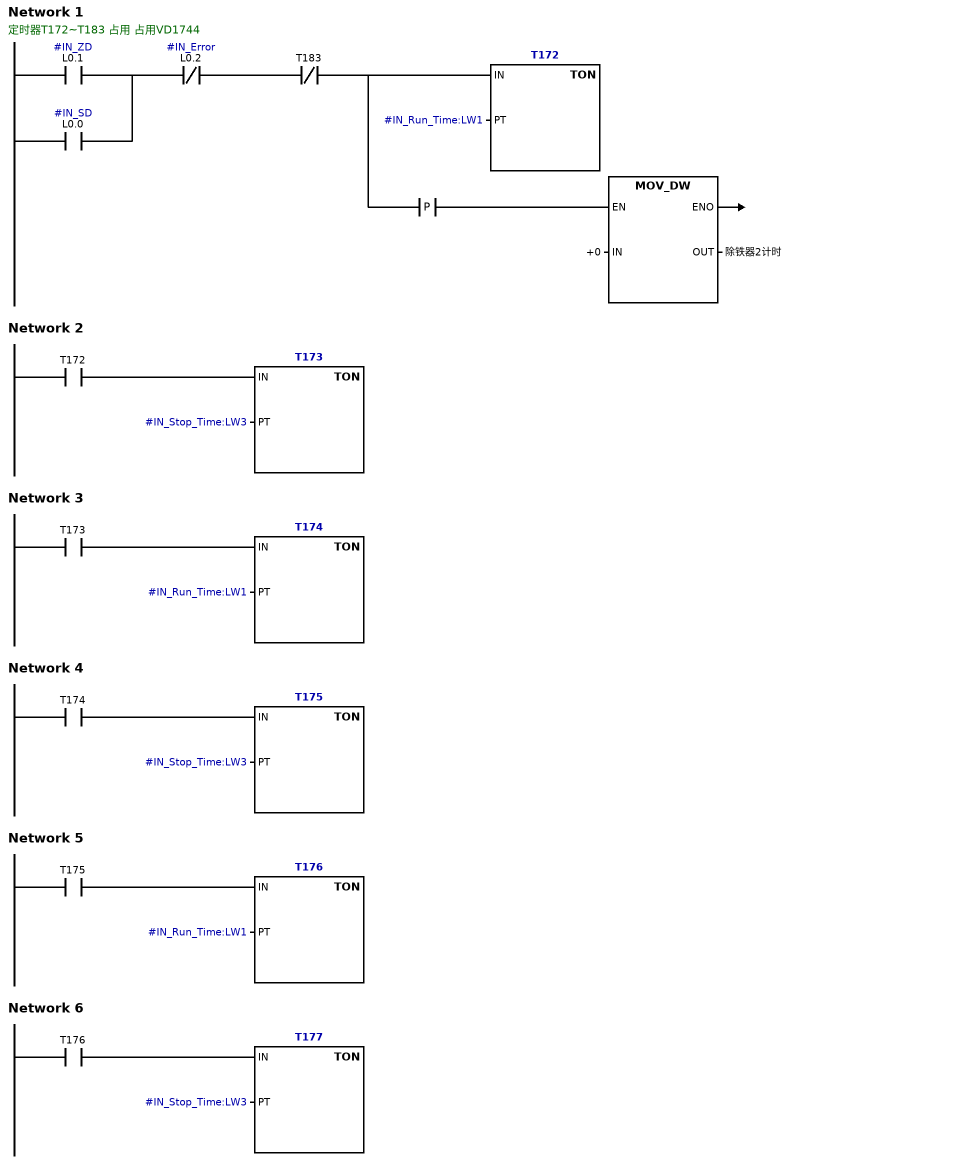
Network 1
// 定时器T172~T183 占用 占用VD1744
// (network saved uncompiled; LAD cells follow)
// row 0: c0 -| |- #IN_ZD:L0.1 v  c1 -|/|- #IN_Error:L0.2  c2 -|/|- T183 v  c3 --  c4 [TON T172 IN:=power@row0, PT:=#IN_Run_Time:LW1]
// row 1: c0 -| |- #IN_SD:L0.0 ^  c2 ^v  c4 [box]
// row 2: c2 ^  c3 -|P|-  c4 --  c5 [MOV_DW EN:=power@row2, IN:=+0, ENO=>power, OUT=>除铁器2计时]  c6 ->
// row 3: c5 [box]
Network 2
LD     T172
TON    T173, #IN_Stop_Time:LW3
Network 3
LD     T173
TON    T174, #IN_Run_Time:LW1
Network 4
LD     T174
TON    T175, #IN_Stop_Time:LW3
Network 5
LD     T175
TON    T176, #IN_Run_Time:LW1
Network 6
LD     T176
TON    T177, #IN_Stop_Time:LW3
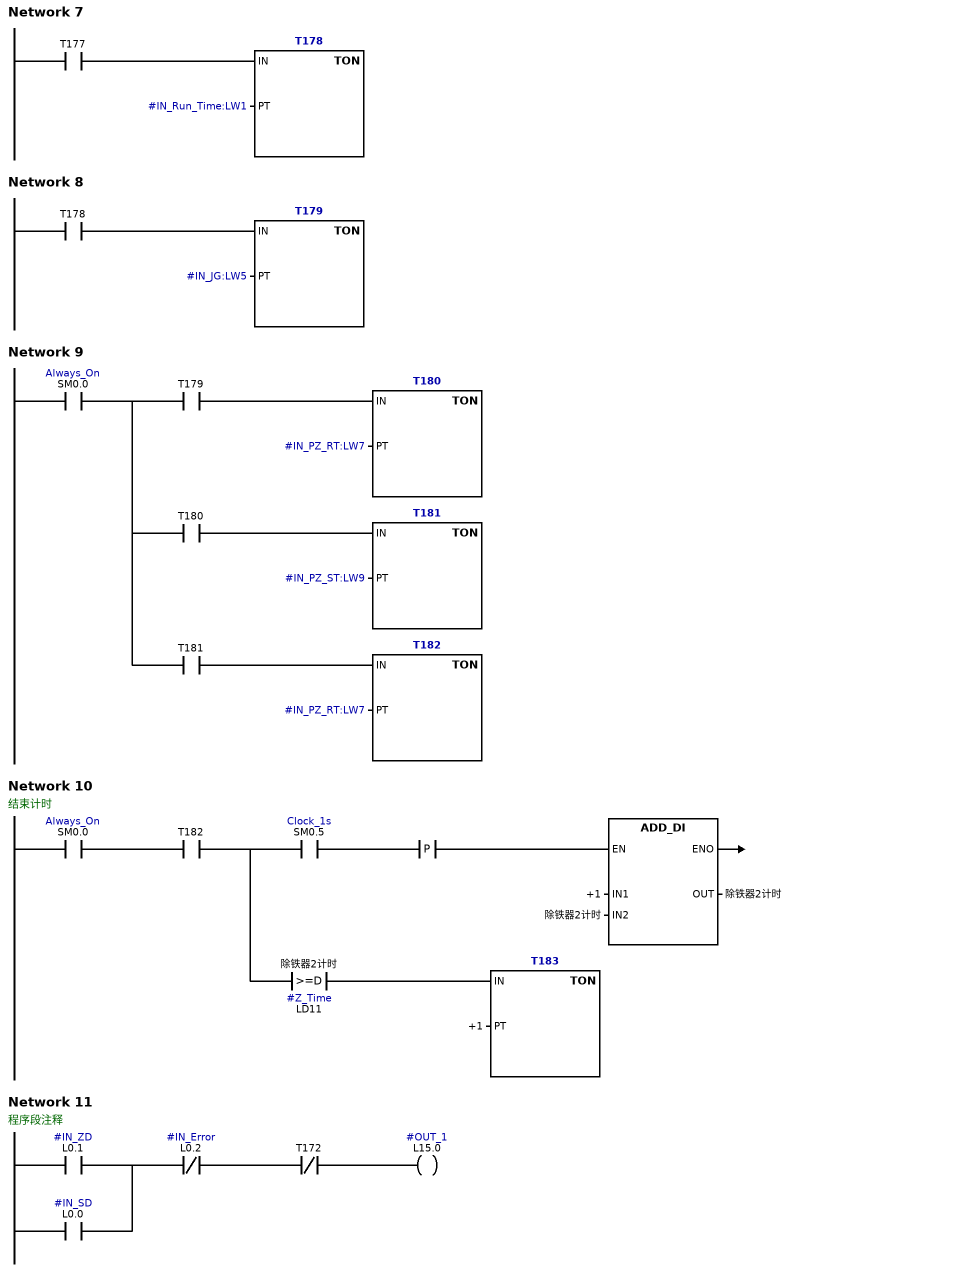
Network 7
LD     T177
TON    T178, #IN_Run_Time:LW1
Network 8
LD     T178
TON    T179, #IN_JG:LW5
Network 9
LD     Always_On:SM0.0
LPS
A      T179
TON    T180, #IN_PZ_RT:LW7
LRD
A      T180
TON    T181, #IN_PZ_ST:LW9
LPP
A      T181
TON    T182, #IN_PZ_RT:LW7
Network 10
// 结束计时
// (network saved uncompiled; LAD cells follow)
// row 0: c0 -| |- Always_On:SM0.0  c1 -| |- T182 v  c2 -| |- Clock_1s:SM0.5  c3 -|P|-  c4 --  c5 [ADD_DI EN:=power@row0, IN1:=+1, IN2:=除铁器2计时, ENO=>power, OUT=>除铁器2计时]  c6 ->
// row 1: c1 ^v  c5 [box]
// row 2: c1 ^  c2 -|>=D|- 除铁器2计时, #Z_Time:LD11  c3 --  c4 [TON T183 IN:=power@row2, PT:=+1]
// row 3: c4 [box]
Network 11
//  程序段注释
LD     #IN_ZD:L0.1
O      #IN_SD:L0.0
AN     #IN_Error:L0.2
AN     T172
=      #OUT_1:L15.0
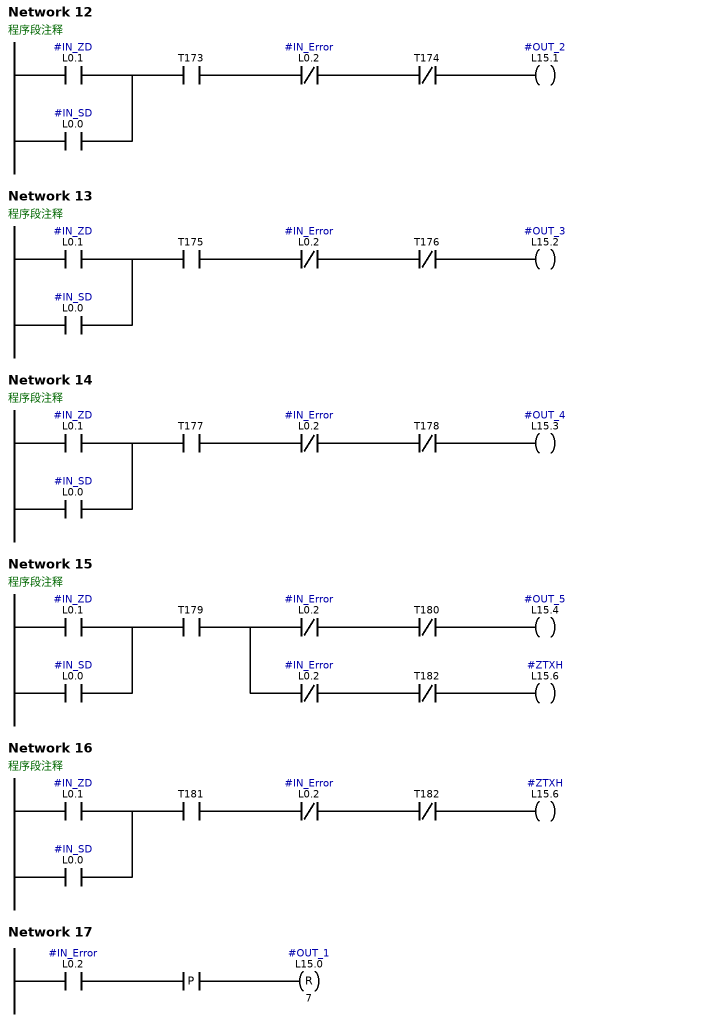
Network 12
//  程序段注释
LD     #IN_ZD:L0.1
O      #IN_SD:L0.0
A      T173
AN     #IN_Error:L0.2
AN     T174
=      #OUT_2:L15.1
Network 13
//  程序段注释
LD     #IN_ZD:L0.1
O      #IN_SD:L0.0
A      T175
AN     #IN_Error:L0.2
AN     T176
=      #OUT_3:L15.2
Network 14
//  程序段注释
LD     #IN_ZD:L0.1
O      #IN_SD:L0.0
A      T177
AN     #IN_Error:L0.2
AN     T178
=      #OUT_4:L15.3
Network 15
//  程序段注释
LD     #IN_ZD:L0.1
O      #IN_SD:L0.0
A      T179
LPS
AN     #IN_Error:L0.2
AN     T180
=      #OUT_5:L15.4
LPP
AN     #IN_Error:L0.2
AN     T182
=      #ZTXH:L15.6
Network 16
//  程序段注释
LD     #IN_ZD:L0.1
O      #IN_SD:L0.0
A      T181
AN     #IN_Error:L0.2
AN     T182
=      #ZTXH:L15.6
Network 17
LD     #IN_Error:L0.2
EU
R      #OUT_1:L15.0, 7
END_SUBROUTINE_BLOCK

SUBROUTINE_BLOCK 除铁器6组3:SBR79
TITLE=
VAR_INPUT
IN_SD:BOOL;	// L0.0 
IN_ZD:BOOL;	// L0.1 
IN_Error:BOOL;	// L0.2 
IN_Run_Time:INT;	// LW1 
IN_Stop_Time:INT;	// LW3 
IN_JG:INT;	// LW5 除铁到排渣间隔
IN_PZ_RT:INT;	// LW7 排渣运行
IN_PZ_ST:INT;	// LW9 排渣间隔
Z_Time:DINT;	// LD11 
END_VAR
VAR_OUTPUT
OUT_1:BOOL;	// L15.0 
OUT_2:BOOL;	// L15.1 
OUT_3:BOOL;	// L15.2 
OUT_4:BOOL;	// L15.3 
OUT_5:BOOL;	// L15.4 
OUT_6:BOOL;	// L15.5 
ZTXH:BOOL;	// L15.6 暂停信号
END_VAR
BEGIN
